// TIA Portal V19 program export: 0 tag tables, 2 data types, 3 data blocks, 8 code blocks (in call order from the OBs), 2 instance data blocks

TYPE "typeCanProcessImageInputs"
   STRUCT
      SlaveDigitalInput1 : Byte;
      SlaveDigitalInput2 : Byte;
      SlaveAnalogInput1 : Int;
      SlaveAnalogInput2 : Int;
      SlaveAnalogInput3 : Int;
      SlaveAnalogInput4 : Int;
   END_STRUCT;
END_TYPE

TYPE "typeCanProcessImageOutputs"
   STRUCT
      SlaveDigitalOutput1 : Byte;
      SlaveDigitalOutput2 : Byte;
      SlaveAnalogOutput1 : Int;
      SlaveAnalogOutput2 : Int;
      SlaveAnalogOutput3 : Int;
      SlaveAnalogOutput4 : Int;
   END_STRUCT;
END_TYPE

DATA_BLOCK "ControlDB"   // DB3
{ S7_Optimized_Access := 'TRUE' }
// stored: MemoryReserve 100
   VAR
      CanProcessImageIn : Array[0..31] of Byte;
      CanProcessImageOut : Array[0..9] of Byte;
      ReadCanProcessImageBusy : Bool;
      ReadCanProcessImageError : Bool;
      ReadCanProcessImageSize : UInt;
      ReadCanProcessImageStatus : DWord;
      ReadCanProcessImageValid : Bool;
      WriteCanProcessImageBusy : Bool;
      WriteCanProcessImageError : Bool;
      WriteCanProcessImageSize : UInt;
      WriteCanProcessImageStatus : DWord;
      WriteCanProcessImageDone : Bool;
      ErrorRegisterReq : Bool;
      ErrorRegisterNode : Int;
      ErrorRegisterBusy : Bool;
      ErrorRegisterGenericError : Bool;
      ErrorRegisterCurrentError : Bool;
      ErrorRegisterVoltageError : Bool;
      ErrorRegisterTemperatureError : Bool;
      ErrorRegisterCommunicationError : Bool;
      ErrorRegisterDeviceSpecificError : Bool;
      ErrorRegisterManufacturerSpecificError : Bool;
      HeartbeatReq : Bool;
      HeartbeatNode : Int;
      HeartbeatMilliseconds : UInt;
      HeartbeatBusy : Bool;
   END_VAR
BEGIN
   CanProcessImageOut[0] := 16#F0;
END_DATA_BLOCK

DATA_BLOCK "MappedCanProcessImageInputs"   // DB9
{ S7_Optimized_Access := 'FALSE' }
   VAR RETAIN
      statCanProcessImageInputs { S7_SetPoint := 'True'} : "typeCanProcessImageInputs";
   END_VAR
BEGIN
END_DATA_BLOCK

DATA_BLOCK "MappedCanProcessImageOutputs"   // DB1
{ S7_Optimized_Access := 'FALSE' }
   VAR RETAIN
      statCanProcessImageOutputs { S7_SetPoint := 'True'} : "typeCanProcessImageOutputs";
   END_VAR
BEGIN
END_DATA_BLOCK

ORGANIZATION_BLOCK "Main"   // OB1, LAD, ProgramCycle
TITLE = "Main Program Sweep (Cycle)"
{ S7_Optimized_Access := 'TRUE' }
// stored: SetENOAutomatically false
   VAR_INPUT
      Initial_Call : Bool;   // Initial call of this OB
      Remanence : Bool;   // =True, if remanent data are available
   END_VAR
BEGIN

REGION Network 1
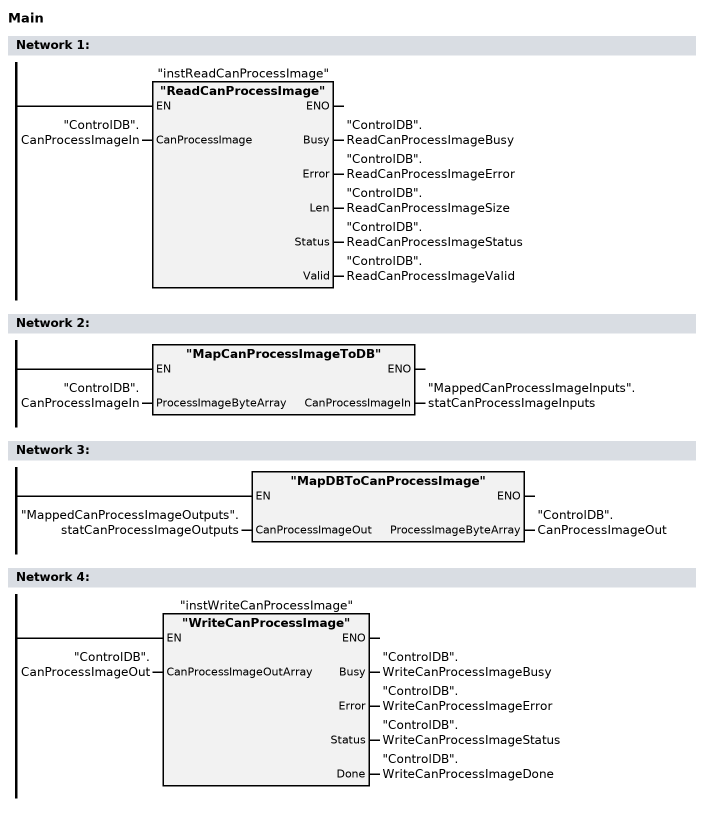
   RUNG wire#powerrail
      "instReadCanProcessImage"(CanProcessImage := "ControlDB".CanProcessImageIn, Busy => "ControlDB".ReadCanProcessImageBusy, Error => "ControlDB".ReadCanProcessImageError, Len => "ControlDB".ReadCanProcessImageSize, Status => "ControlDB".ReadCanProcessImageStatus, Valid => "ControlDB".ReadCanProcessImageValid)
   END_RUNG
   // the same network as SCL:
   "instReadCanProcessImage"(CanProcessImage := "ControlDB".CanProcessImageIn,   // "ReadCanProcessImage"
                           Busy => "ControlDB".ReadCanProcessImageBusy,
                           Error => "ControlDB".ReadCanProcessImageError,
                           Len => "ControlDB".ReadCanProcessImageSize,
                           Status => "ControlDB".ReadCanProcessImageStatus,
                           Valid => "ControlDB".ReadCanProcessImageValid);
END_REGION

REGION Network 2
   RUNG wire#powerrail
      "MapCanProcessImageToDB"(ProcessImageByteArray := "ControlDB".CanProcessImageIn, CanProcessImageIn => "MappedCanProcessImageInputs".statCanProcessImageInputs)
   END_RUNG
   // the same network as SCL:
   "MapCanProcessImageToDB"(ProcessImageByteArray := "ControlDB".CanProcessImageIn,
                           CanProcessImageIn => "MappedCanProcessImageInputs".statCanProcessImageInputs);
END_REGION

REGION Network 3
   RUNG wire#powerrail
      "MapDBToCanProcessImage"(CanProcessImageOut := "MappedCanProcessImageOutputs".statCanProcessImageOutputs, ProcessImageByteArray => "ControlDB".CanProcessImageOut)
   END_RUNG
   // the same network as SCL:
   "MapDBToCanProcessImage"(CanProcessImageOut := "MappedCanProcessImageOutputs".statCanProcessImageOutputs,
                           ProcessImageByteArray => "ControlDB".CanProcessImageOut);
END_REGION

REGION Network 4
   RUNG wire#powerrail
      "instWriteCanProcessImage"(CanProcessImageOutArray := "ControlDB".CanProcessImageOut, Busy => "ControlDB".WriteCanProcessImageBusy, Error => "ControlDB".WriteCanProcessImageError, Status => "ControlDB".WriteCanProcessImageStatus, Done => "ControlDB".WriteCanProcessImageDone)
   END_RUNG
   // the same network as SCL:
   "instWriteCanProcessImage"(CanProcessImageOutArray := "ControlDB".CanProcessImageOut,   // "WriteCanProcessImage"
                           Busy => "ControlDB".WriteCanProcessImageBusy,
                           Error => "ControlDB".WriteCanProcessImageError,
                           Status => "ControlDB".WriteCanProcessImageStatus,
                           Done => "ControlDB".WriteCanProcessImageDone);
END_REGION
END_ORGANIZATION_BLOCK

FUNCTION_BLOCK "ReadCanProcessImage"
{ S7_Optimized_Access := 'TRUE' }
VERSION : 0.1
   VAR_OUTPUT 
      Busy : Bool;
      Error : Bool;
      Len : UInt;
      Status : DWord;
      Valid : Bool;
   END_VAR

   VAR_IN_OUT 
      CanProcessImage : Array[0..31] of Byte;
   END_VAR


BEGIN
	    "RDREC_DB"(REQ := true,
	               ID := 269,
	               INDEX := 16#90,
	               MLEN := 32,
	               RECORD := #CanProcessImage,
	               BUSY => #Busy,
	               ERROR => #Error,
	               LEN => #Len,
	               STATUS => #Status,
	               VALID => #Valid);
	    
	// It might be an issue that REQ is always true since it uses a rising edge
	// according to ChatGPT. I haven't noticed any issues.
	    
	// (written by Siemens dev for application example, not sure what it's for)
	// IF #Valid = true  THEN
	//     "ControlDB".Read := false;
	// END_IF;
	
END_FUNCTION_BLOCK

FUNCTION "MapCanProcessImageToDB" : Void
{ S7_Optimized_Access := 'TRUE' }
VERSION : 0.1
   VAR_INPUT 
      ProcessImageByteArray : Array[0..31] of Byte;
   END_VAR

   VAR_IN_OUT 
      CanProcessImageIn : "typeCanProcessImageInputs";
   END_VAR


BEGIN
	// Double buffer functionality implemented for asynchronous access (snap7)
	IF #CanProcessImageIn.ActiveBuffer = 0 THEN
	    //map bytes 
	    #CanProcessImageIn.BufferB.SlaveDigitalInput1 := #ProcessImageByteArray[0];
	    #CanProcessImageIn.BufferB.SlaveDigitalInput2 := #ProcessImageByteArray[1];
	    
	    //map words
	    #CanProcessImageIn.BufferB.SlaveAnalogInput1 := "BytesToWord"(Byte0 := #ProcessImageByteArray[2], Byte1 := #ProcessImageByteArray[3]);
	    #CanProcessImageIn.BufferB.SlaveAnalogInput2 := "BytesToWord"(Byte0 := #ProcessImageByteArray[4], Byte1 := #ProcessImageByteArray[5]);
	    #CanProcessImageIn.BufferB.SlaveAnalogInput3 := "BytesToWord"(Byte0 := #ProcessImageByteArray[6], Byte1 := #ProcessImageByteArray[7]);
	    #CanProcessImageIn.BufferB.SlaveAnalogInput4 := "BytesToWord"(Byte0 := #ProcessImageByteArray[8], Byte1 := #ProcessImageByteArray[9]);
	    
	    #CanProcessImageIn.ActiveBuffer := 1;
	ELSE
	    //map bytes 
	    #CanProcessImageIn.BufferA.SlaveDigitalInput1 := #ProcessImageByteArray[0];
	    #CanProcessImageIn.BufferA.SlaveDigitalInput2 := #ProcessImageByteArray[1];
	    
	    //map words
	    #CanProcessImageIn.BufferA.SlaveAnalogInput1 := "BytesToWord"(Byte0 := #ProcessImageByteArray[2], Byte1 := #ProcessImageByteArray[3]);
	    #CanProcessImageIn.BufferA.SlaveAnalogInput2 := "BytesToWord"(Byte0 := #ProcessImageByteArray[4], Byte1 := #ProcessImageByteArray[5]);
	    #CanProcessImageIn.BufferA.SlaveAnalogInput3 := "BytesToWord"(Byte0 := #ProcessImageByteArray[6], Byte1 := #ProcessImageByteArray[7]);
	    #CanProcessImageIn.BufferA.SlaveAnalogInput4 := "BytesToWord"(Byte0 := #ProcessImageByteArray[8], Byte1 := #ProcessImageByteArray[9]);
	    
	    #CanProcessImageIn.ActiveBuffer := 0;
	END_IF;
	
	
	//map dwords
	// Byte order reversed in application example. Not sure why as the expected byte order worked fine for me; change order as needed.
	
	// There aren't any dwords in use in the current program, but here is an example if needed in the future:
	// #CanProcessImageIn.SensorInPvTemperature := "BytesToDoubleWord"(Byte0 :=#ProcessImageByteArray[11],
	//                  Byte1 :=#ProcessImageByteArray[10],
	//                  Byte2 :=#ProcessImageByteArray[9],
	//                  Byte3 :=#ProcessImageByteArray[8]);
	//                  
	
	// To avoid using functions for this process, use slice notation:
	//     #CanProcessImageIn.SlaveAnalogInput1.%B0 := #ProcessImageByteArray[3]; // Low byte
	//     #CanProcessImageIn.SlaveAnalogInput1.%B1 := #ProcessImageByteArray[2]; // High byte
	
END_FUNCTION

FUNCTION "BytesToWord" : Word
{ S7_Optimized_Access := 'TRUE' }
VERSION : 0.1
   VAR_INPUT 
      Byte0 : Byte;
      Byte1 : Byte;
   END_VAR


BEGIN
	//This block turns two bytes into a word (little-endian)
	//The order of bytes within the resulting word is: B1B0
	
	//Example: Byte0 is 1111111 and Byte1 is 10101010
	//This operation will add Byte0 (1111111) to the 8-bit-leftshifted version of Byte1 (10101010 00000000)
	//10101010 00000000 + 11111111
	//Result Word = 10101010 11111111
	#BytesToWord := BYTE_TO_WORD(IN:=#Byte0) + SHL(IN := BYTE_TO_WORD(IN:=#Byte1), N := 8);
END_FUNCTION

FUNCTION "BytesToDoubleWord" : DWord
{ S7_Optimized_Access := 'TRUE' }
VERSION : 0.1
   VAR_INPUT 
      Byte0 : Byte;
      Byte1 : Byte;
      Byte2 : Byte;
      Byte3 : Byte;
   END_VAR

   VAR_TEMP 
      tempWord0 : Word;
      tempWord1 : Word;
   END_VAR


BEGIN
	//This function block creates a Dword out of four bytes
	//The order of bytes within the resulting Dword is: B3B2B1B0
	
	
	#tempWord0:= "BytesToWord"(Byte0 := #Byte0, Byte1 := #Byte1);
	#tempWord1 := "BytesToWord"(Byte0 := #Byte2, Byte1 := #Byte3);
	
	#BytesToDoubleWord := WORD_TO_DWORD(IN:=#tempWord0) + SHL(IN := WORD_TO_DWORD(IN:=#tempWord1), N := 16);
	
	
END_FUNCTION

FUNCTION_BLOCK "WriteCanProcessImage"
{ S7_Optimized_Access := 'TRUE' }
VERSION : 0.1
   VAR_OUTPUT 
      Busy : Bool;
      Error : Bool;
      Status : DWord;
      Done : Bool;
   END_VAR

   VAR_IN_OUT 
      CanProcessImageOutArray : Array[0..9] of Byte;
   END_VAR


BEGIN
	
	    "WRREC_DB"(REQ := true,
	               ID := 269,
	               INDEX := 16#91,
	               LEN := 10,
	               DONE => #Done,
	               BUSY => #Busy,
	               ERROR => #Error,
	               STATUS => #Status,
	               RECORD := #CanProcessImageOutArray);
	    
	// Changed len from 4 to 10 since my output process image is larger now. Also changed the InOut variable's array size
	
	// IF #Done = true  THEN
	//     "ControlDB".Write := false;
	// END_IF;
	
END_FUNCTION_BLOCK

FUNCTION "InvertWordEndianness" : Word
{ S7_Optimized_Access := 'FALSE' }
VERSION : 0.1
   VAR_INPUT 
      InputWord : Word;
   END_VAR

   VAR_TEMP 
      tempInputByte0 : Byte;
      tempInputByte1 : Byte;
   END_VAR


BEGIN
	#tempInputByte0 := WORD_TO_BYTE(#InputWord & 2#0000000011111111); // Least significant portion of word (little-endian)
	#tempInputByte1 := WORD_TO_BYTE(SHR(IN:=#InputWord, N:=8));       // Most significant portion of word (little-endian)  
	
	// I believe this code is incorrect. #tempInputByte0 and #tempInputByte1 should be swapped to invert the endianness
	#InvertWordEndianness := "BytesToWord"(Byte0 := #tempInputByte0, Byte1 := #tempInputByte1);
	
END_FUNCTION

FUNCTION "WordToBytes" : Void
{ S7_Optimized_Access := 'TRUE' }
VERSION : 0.1
   VAR_INPUT 
      "Word" : Word;
   END_VAR

   VAR_OUTPUT 
      Byte0 : Byte;
      Byte1 : Byte;
   END_VAR


BEGIN
	#Byte0 := WORD_TO_BYTE(#Word AND 2#0000000011111111);
	#Byte1 := WORD_TO_BYTE(SHR(IN := #Word, N := 8));
END_FUNCTION

DATA_BLOCK "instReadCanProcessImage"   // DB5
// stored: AutoNumber false, InstanceOfName ReadCanProcessImage, InstanceOfType FB
"ReadCanProcessImage"
BEGIN
END_DATA_BLOCK

DATA_BLOCK "instWriteCanProcessImage"   // DB16
// stored: AutoNumber false, InstanceOfName WriteCanProcessImage, InstanceOfType FB
"WriteCanProcessImage"
BEGIN
END_DATA_BLOCK
